FUNCTION_BLOCK PAFDischarging EXTENDS PARoutingFunction IMPLEMENTS IPAFDischarging
VAR_INPUT
END_VAR
VAR_OUTPUT
END_VAR
VAR
	_ACMethod : ACMethodDischarging;
	_StateTolerance : PANotifyState;	
	_FaultAckTolerance : BOOL;
	_StateDestinationFull : PANotifyState;	
	_FaultAckDestinationFull : BOOL;
END_VAR

PROPERTY ACMethod : IACMethod
GET
ACMethod := _ACMethod;
END_GET
END_PROPERTY

{attribute 'TcRpcEnable'}
PROPERTY PUBLIC FaultAckDestinationFull : BOOL
GET
FaultAckDestinationFull := _FaultAckDestinationFull;
END_GET
SET
_FaultAckDestinationFull := FaultAckDestinationFull;
Root.OnPropertyChangedBool(THIS^, 22, _FaultAckDestinationFull);
END_SET
END_PROPERTY

{attribute 'TcRpcEnable'}
PROPERTY PUBLIC FaultAckTolerance : BOOL
GET
FaultAckTolerance := _FaultAckTolerance;
END_GET
SET
_FaultAckTolerance := FaultAckTolerance;
Root.OnPropertyChangedBool(THIS^, 20, _FaultAckTolerance);
END_SET
END_PROPERTY

METHOD PUBLIC FB_postinit
VAR_INPUT
	root : IACVariobatch;
END_VAR
SUPER^.FB_postinit(root);
root.OnPropertyChangedInt(THIS^, 19, _StateTolerance);
root.OnPropertyChangedBool(THIS^, 20, _FaultAckTolerance);
root.OnPropertyChangedInt(THIS^, 21, _StateDestinationFull);
root.OnPropertyChangedBool(THIS^, 22, _FaultAckDestinationFull);
END_METHOD

METHOD OnInitMemory
VAR_INPUT
		root : IACVariobatch;	
END_VAR
RegisterProperty(root, 19, GCL.cSizeINT); //_StateTolerance)
RegisterProperty(root, 20, GCL.cSizeBYTE); //_FaultAckTolerance);
RegisterProperty(root, 21, GCL.cSizeINT); //_StateDestinationFull)
RegisterProperty(root, 22, GCL.cSizeBYTE); //_FaultAckDestinationFull);
SUPER^.OnInitMemory(root);
END_METHOD

METHOD PUBLIC InvokeSetterEnum
VAR_INPUT
	PropertyID : INT;
	PropertyValue : INT;
END_VAR
SUPER^.InvokeSetterEnum(PropertyID, PropertyValue);
IF PropertyID = 19 THEN
	THIS^.StateTolerance := PropertyValue;
ELSIF PropertyID = 21 THEN	
	THIS^.StateDestinationFull := PropertyValue;
END_IF
END_METHOD

METHOD PROTECTED SMIdle
VAR_INPUT
END_VAR
SUPER^.SMIdle();
END_METHOD

METHOD PUBLIC StartWithP : BOOL
VAR_INPUT
	parameter : ACMethodDischargingP;
END_VAR
VAR
	acMethod : ACMethodDischarging;
END_VAR
acMethod.Parameter := parameter;
_ACMethod.ResolveRoutePointers(parameter._Route, THIS^);
IF NOT acMethod.IsValid THEN
		StartWithP := FALSE;
	RETURN;
END_IF
_ACMethod.Parameter := parameter;
StartWithP := Start();
END_METHOD

PROPERTY PUBLIC StateDestinationFull : PANotifyState
GET
StateDestinationFull := _StateDestinationFull;
END_GET
SET
_StateDestinationFull := StateDestinationFull;
Root.OnPropertyChangedInt(THIS^, 21, _StateDestinationFull);
END_SET
END_PROPERTY

PROPERTY PUBLIC StateTolerance : PANotifyState
GET
StateTolerance := _StateTolerance;
END_GET
SET
_StateTolerance := StateTolerance;
Root.OnPropertyChangedInt(THIS^, 19, _StateTolerance);
END_SET
END_PROPERTY

END_FUNCTION_BLOCK

(* stored: Version 1.1.0.1, ProductVersion 3.1.4020.12
   POU PAFDischarging: Id {a9a63cc6-1b38-45da-bfd0-ac924af755fc}, SpecialFunc None
   Folder Properties: Id {2cc58cb4-1fd8-4b64-ba31-eb91854a6033}
   Folder StateMethods: Id {a80b371d-1c0a-474f-8200-0cd4a82be6ce}
   Property ACMethod: Id {de3f4728-a635-4105-bfe8-bafbf47552eb}
   Get Get: Id {7d6165ab-1a01-4caa-87ff-9cd02cc71721}
   Property FaultAckDestinationFull: Id {818ed8ec-9a07-4603-8862-dfae7a6309ff}
   Get Get: Id {6ee456d7-4a72-4bac-b0d6-1c47ebe39323}
   Set Set: Id {668546a6-a464-441b-a059-12f02b57bfd0}
   Property FaultAckTolerance: Id {4142ad06-2d2c-40cc-bb68-0e0b7d493607}
   Get Get: Id {f3eb2ac2-8b8c-4f42-88eb-245d0adb9a7e}
   Set Set: Id {2991023f-42ec-4ecc-8bbb-81dc0258d7b3}
   Method FB_postinit: Id {4d7c2572-5675-460c-a274-0cc99e2ef780}
   Method OnInitMemory: Id {b6f3cf6e-0ab7-4073-a8ce-f1fd8c22add2}
   Method InvokeSetterEnum: Id {786f492b-1112-4d0a-a754-1fe1e5d34a72}
   Method SMIdle: Id {d3b38740-7db4-47b8-b20d-093a85d38892}
   Method StartWithP: Id {06ebd9f0-e50c-4825-a347-2082481c3436}
   Property StateDestinationFull: Id {dfa58686-0e6e-490b-934d-77131c61ef8c}
   Get Get: Id {43198cb6-6b53-4160-a987-b3544be3d883}
   Set Set: Id {72fdb225-759b-4077-b038-3fb23bb15799}
   Property StateTolerance: Id {1ceb5c08-ae26-4d4f-9252-6e006db56d7d}
   Get Get: Id {933d39ba-83f3-4a07-8e2e-8316510d3a33}
   Set Set: Id {fcfbfe38-7165-4cbd-a9dd-e71da2b352b0} *)
